// TwinCAT 3 PLC project Resolver_Test_Rig_Program
// ProgramVersion: 3.1.4023.0
// libraries:
//   Tc2_MC2, * (Beckhoff Automation GmbH)
//   Tc2_Standard, * (Beckhoff Automation GmbH)
//   Tc2_System, * (Beckhoff Automation GmbH)
//   Tc2_Utilities, * (Beckhoff Automation GmbH)
//   Tc3_Module, * (Beckhoff Automation GmbH)
//   VisuDialogs, * (System)
// project tree:
//   DUTs/ DUT_fileWriterStates.TcDUT, ST_EncoderCSVData.TcDUT
//   / GlobalTextList.TcGTLO, PlcTask.TcTTO, Visualization Manager.TcVMO (not stored)
//   GVLs/ GVL.TcGVL
//   POUs/ MAIN.TcPOU, FB_Stage_Motion.TcPOU, P_CSVWriter.TcPOU
//   POUs/UnixTimestamp/ UnixTimestamp.TcPOU (not stored)
//   VISUs/ Alarms.TcVIS, Manual_Operations.TcVIS, Run_Screen.TcVIS, Set_Up.TcVIS, Visualization.TcVIS
// real-time tasks:
//   TASK PlcTask: cycle T#10ms, priority 5, ADS port 350
// motion (NC):
//   TASK NC-Task 1 SAF: cycle T#2ms, priority 4, ADS port 501
//   TASK NC-Task 1 SVB: cycle T#10ms, priority 8, ADS port 511
//   AXIS Axis 1 (id 1)
//     Dynamic: AccelerationMaximum=375, DecelerationMaximum=375
//     Velo: SlowManual=0.5, FastManual=1, Maximum=50
//     OtherSettings: AllowMotionCmdToSlave=true
//     encoder EncType=4
//       EncPara: ScaleFactorNumerator=0.00015625, MaxCount=#x0000ffff
//         Inc: RefMode=2, RefSoftSyncMask=#x0000ffff
//     drive DrvType=24
//       Analog: VeloReferenz=20, TorqueScale=10, ScaleFactorActTorque=0.1
//       TimeComp: TaskDelayCycles=1
//     controller CtrType=1
//       CtrPara: PriorControlFactor=1
//         Observer: BandWidth=20
//   AXIS Axis 2 (id 2)
//     OtherSettings: AllowMotionCmdToSlave=true
//     encoder EncType=5
//       EncPara: ScaleFactorNumerator=0.5, ScaleFactorDenominator=65536, MaxCount=#xffffffff, ReferenceSystem=1
//     drive DrvType=5
//       Analog: TorqueScale=10, ScaleFactorActTorque=0.1
//       TimeComp: TaskDelayCycles=1
//     controller CtrType=1
//       CtrPara: PriorControlFactor=1
//         Observer: BandWidth=20
//   AXIS Axis 3 (id 3)
//     OtherSettings: AllowMotionCmdToSlave=true
//     encoder EncType=5
//       EncPara: ScaleFactorNumerator=2, ScaleFactorDenominator=4096, ReferenceSystem=1
//     drive DrvType=5
//       Analog: TorqueScale=10, ScaleFactorActTorque=0.1
//       TimeComp: TaskDelayCycles=1
//     controller CtrType=1
//       CtrPara: PriorControlFactor=1
//         Observer: BandWidth=20
//   AXIS Axis 4 (id 4)
//     OtherSettings: AllowMotionCmdToSlave=true
//     encoder EncType=29
//       EncPara: MaxCount=#xffffffff
//     drive DrvType=5
//       Analog: TorqueScale=10, ScaleFactorActTorque=0.1
//       TimeComp: TaskDelayCycles=1
//     controller CtrType=1
//       CtrPara: PriorControlFactor=1
//         Observer: BandWidth=20
// I/O:
//   DEVICE Device 1 (EtherCAT) (disabled), AmsNetId 130.246.57.106.2.1
//     Term 8 (EK1200) [EK1200-5000 EtherCAT Power supply (2A E-Bus)]
//       Term 9 (EL1008) [EL1008 8Ch. Dig. Input 24V, 3ms]
//       Term 10 (EL2808) [EL2808 8Ch. Dig. Output 24V, 0.5A]
//       Term 11 (EL7047) [EL7047 1Ch. Stepper motor output stage (50V, 5A)]
//       Term 12 (EL5002) [EL5002 2Ch. SSI Encoder]
//       Term 1 (EL5042) [EL5042 2Ch. BiSS-C Encoder]
//       Term 2 (EL3314-0002) [EL3314-0002 4Ch. Ana Input Thermocouple (TC), Isolated Channels]
//       Term 13 (EL9011) [EL9011 End Terminal]
// variable links:
//   NC-Task 1 SAF/Axes/Axis 1 <-> Device 1 (EtherCAT)/Term 8 (EK1200)/Term 11 (EL7047)
//     Drive/Inputs/In/nState1 @bit 3 <-> STM Status/Status/Error
//     Drive/Inputs/In/nState1 @bit 7 <-> STM Status/Status/Motor stall
//     Drive/Inputs/In/nState1 @bit 5 <-> STM Status/Status/Moving negative
//     Drive/Inputs/In/nState1 @bit 4 <-> STM Status/Status/Moving positive
//     Drive/Inputs/In/nState1 @bit 1 <-> STM Status/Status/Ready
//     Drive/Inputs/In/nState1 <-> STM Status/Status/Ready to enable
//     Drive/Inputs/In/nState1 @bit 6 <-> STM Status/Status/Torque reduced
//     Drive/Inputs/In/nState1 @bit 2 <-> STM Status/Status/Warning
//     Drive/Inputs/In/nState2 @bit 3 <-> STM Status/Status/Digital input 1
//     Drive/Inputs/In/nState2 @bit 4 <-> STM Status/Status/Digital input 2
//     Drive/Inputs/In/nState2 @bit 5 <-> STM Status/Status/Sync error
//     Drive/Inputs/In/nState2 @bit 7 <-> STM Status/Status/TxPDO Toggle
//     Drive/Inputs/In/nState4 @bit 1 <-> WcState/InputToggle
//     Drive/Inputs/In/nState4 <-> WcState/WcState
//     Drive/Outputs/Out/nCtrl1 <-> STM Control/Control/Enable
//     Drive/Outputs/Out/nCtrl1 @bit 2 <-> STM Control/Control/Reduce torque
//     Drive/Outputs/Out/nCtrl1 @bit 1 <-> STM Control/Control/Reset
//     Drive/Outputs/Out/nCtrl2 @bit 3 <-> STM Control/Control/Digital output 1
//     Drive/Outputs/Out/nDataOut2[0] <-> STM Velocity/Velocity
//     Enc/Inputs/In/nDataIn1[0] <-> ENC Status compact/Counter value
//     Enc/Inputs/In/nDataIn2[0] <-> ENC Status compact/Latch value
//     Enc/Inputs/In/nState1 @bit 4 <-> ENC Status compact/Status/Counter overflow
//     Enc/Inputs/In/nState1 @bit 3 <-> ENC Status compact/Status/Counter underflow
//     Enc/Inputs/In/nState1 @bit 7 <-> ENC Status compact/Status/Extrapolation stall
//     Enc/Inputs/In/nState1 <-> ENC Status compact/Status/Latch C valid
//     Enc/Inputs/In/nState1 @bit 1 <-> ENC Status compact/Status/Latch extern valid
//     Enc/Inputs/In/nState1 @bit 2 <-> ENC Status compact/Status/Set counter done
//     Enc/Inputs/In/nState2 @bit 4 <-> ENC Status compact/Status/Status of extern latch
//     Enc/Inputs/In/nState2 <-> ENC Status compact/Status/Status of input A
//     Enc/Inputs/In/nState2 @bit 1 <-> ENC Status compact/Status/Status of input B
//     Enc/Inputs/In/nState2 @bit 2 <-> ENC Status compact/Status/Status of input C
//     Enc/Inputs/In/nState2 @bit 5 <-> ENC Status compact/Status/Sync error
//     Enc/Inputs/In/nState2 @bit 7 <-> ENC Status compact/Status/TxPDO Toggle
//     Enc/Inputs/In/nState4 @bit 1 <-> WcState/InputToggle
//     Enc/Inputs/In/nState4 <-> WcState/WcState
//     Enc/Outputs/Out/nCtrl1 <-> ENC Control compact/Control/Enable latch C
//     Enc/Outputs/Out/nCtrl1 @bit 3 <-> ENC Control compact/Control/Enable latch extern on negative edge
//     Enc/Outputs/Out/nCtrl1 @bit 1 <-> ENC Control compact/Control/Enable latch extern on positive edge
//     Enc/Outputs/Out/nCtrl1 @bit 2 <-> ENC Control compact/Control/Set counter
//     Enc/Outputs/Out/nDataOut1[0] <-> ENC Control compact/Set counter value
//   NC-Task 1 SAF/Axes/Axis 2 <-> Device 1 (EtherCAT)/Term 8 (EK1200)/Term 12 (EL5002)
//     Enc/Inputs/In/nDataIn1 <-> SSI Inputs Channel 1/Counter value
//     Enc/Inputs/In/nState1 <-> SSI Inputs Channel 1/Status/Data error
//     Enc/Inputs/In/nState1 @bit 3 <-> SSI Inputs Channel 1/Status/Data mismatch
//     Enc/Inputs/In/nState1 @bit 1 <-> SSI Inputs Channel 1/Status/Frame error
//     Enc/Inputs/In/nState1 @bit 2 <-> SSI Inputs Channel 1/Status/Power failure
//     Enc/Inputs/In/nState2 @bit 5 <-> SSI Inputs Channel 1/Status/Sync error
//     Enc/Inputs/In/nState2 @bit 6 <-> SSI Inputs Channel 1/Status/TxPDO State
//     Enc/Inputs/In/nState2 @bit 7 <-> SSI Inputs Channel 1/Status/TxPDO Toggle
//     Enc/Inputs/In/nState4 @bit 1 <-> WcState/InputToggle
//     Enc/Inputs/In/nState4 <-> WcState/WcState
//   NC-Task 1 SAF/Axes/Axis 3 <-> Device 1 (EtherCAT)/Term 8 (EK1200)/Term 12 (EL5002)
//     Enc/Inputs/In/nDataIn1 <-> SSI Inputs Channel 2/Counter value
//     Enc/Inputs/In/nState1 <-> SSI Inputs Channel 2/Status/Data error
//     Enc/Inputs/In/nState1 @bit 3 <-> SSI Inputs Channel 2/Status/Data mismatch
//     Enc/Inputs/In/nState1 @bit 1 <-> SSI Inputs Channel 2/Status/Frame error
//     Enc/Inputs/In/nState1 @bit 2 <-> SSI Inputs Channel 2/Status/Power failure
//     Enc/Inputs/In/nState2 @bit 5 <-> SSI Inputs Channel 2/Status/Sync error
//     Enc/Inputs/In/nState2 @bit 6 <-> SSI Inputs Channel 2/Status/TxPDO State
//     Enc/Inputs/In/nState2 @bit 7 <-> SSI Inputs Channel 2/Status/TxPDO Toggle
//     Enc/Inputs/In/nState4 @bit 1 <-> WcState/InputToggle
//     Enc/Inputs/In/nState4 <-> WcState/WcState
//   NC-Task 1 SAF/Axes/Axis 4 <-> Device 1 (EtherCAT)/Term 8 (EK1200)/Term 1 (EL5042)
//     Enc/Inputs/In/nComState @bit 1 <-> WcState/InputToggle
//     Enc/Inputs/In/nComState <-> WcState/WcState
//     Enc/Inputs/In/nDataIn1 <-> FB Inputs Channel 1/Position
//     Enc/Inputs/In/nState1 @bit 12 <-> FB Inputs Channel 1/Status/Diag
//     Enc/Inputs/In/nState1 @bit 1 <-> FB Inputs Channel 1/Status/Error
//     Enc/Inputs/In/nState1 @bit 14 <-> FB Inputs Channel 1/Status/Input cycle counter
//     Enc/Inputs/In/nState1 @bit 2 <-> FB Inputs Channel 1/Status/Ready
//     Enc/Inputs/In/nState1 @bit 13 <-> FB Inputs Channel 1/Status/TxPDO State
//     Enc/Inputs/In/nState1 <-> FB Inputs Channel 1/Status/Warning
//   Resolver_Test_Rig_Program/Resolver_Test_Rig_Program Instance <-> Device 1 (EtherCAT)/Term 8 (EK1200)/Term 10 (EL2808)
//     PlcTask Outputs/MAIN.EncoderPowerOutput_3 <-> Channel 3/Output
//     PlcTask Outputs/MAIN.EncoderPowerOutput_6 <-> Channel 6/Output
//     PlcTask Outputs/MAIN.LimitSwitchOutput_1 <-> Channel 1/Output
//     PlcTask Outputs/MAIN.LimitSwitchOutput_2 <-> Channel 2/Output
//   Resolver_Test_Rig_Program/Resolver_Test_Rig_Program Instance <-> Device 1 (EtherCAT)/Term 8 (EK1200)/Term 9 (EL1008)
//     PlcTask Inputs/MAIN.LimitSwitchInput_1 <-> Channel 1/Input
//     PlcTask Inputs/MAIN.LimitSwitchInput_2 <-> Channel 2/Input

CONFIGURATION Resolver_Test_Rig_Program
    RESOURCE PLC ON TwinCAT3
        TASK PlcTask(INTERVAL := T#10ms, PRIORITY := 5);
        PROGRAM MAIN WITH PlcTask : MAIN;
    END_RESOURCE
END_CONFIGURATION

// ---- DUTs/DUT_fileWriterStates.TcDUT
{attribute 'qualified_only'}
{attribute 'strict'}
TYPE DUT_fileWriterStates :
(
	
    idle := 0,
    opening,
    saving,
    closing,
    error

);
END_TYPE

// ---- DUTs/ST_EncoderCSVData.TcDUT
TYPE ST_EncoderCSVData :
STRUCT
	MeasurementID           : INT;
    testState               : INT;
    AxisPosition            : LREAL;
    CurrentCycle            : WORD;
    PositalPosition         : LREAL;
    KublerPosition          : LREAL;
    AMOPosition             : REAL;
    ThermoCouple            : ARRAY[0..3] OF DINT;
    UnixTime                : ULINT;
END_STRUCT
END_TYPE

// ---- GVLs/GVL.TcGVL
{attribute 'Tc2GvlVarNames'}
VAR_GLOBAL CONSTANT
	

	MAX_CSV_ROWS             : UDINT := 1;
    MAX_CSV_COLUMNS         : UDINT := 12;
    MAX_CSV_FIELD_LENGTH    : UDINT := 100;
   
    DATA_CSV_HEADERS        : ARRAY[0..MAX_CSV_COLUMNS] OF STRING(MAX_CSV_FIELD_LENGTH) :=[ (* Source PLC database *)
    'MeasurementID',
    'TestState',
    'AxisPosition',
    'CurrentCycle',
    'PositalPosition',
    'KublerPosition',
    'AMOPosition',
    'ThermoCouple_1',
    'ThermoCouple_2',
    'ThermoCouple_3',
    'ThermoCouple_4',  
    'UnixTime']; 

END_VAR 
VAR_GLOBAL
		stAxis_1 : AXIS_REF;
		stAxis_2 : AXIS_REF;
		stAxis_3 : AXIS_REF;
		stAxis_4 : AXIS_REF;
		

END_VAR

// ---- POUs/MAIN.TcPOU
PROGRAM MAIN
VAR
		// stepper function blocks  
	mcPower_1 : MC_Power;
	mcReset_1 : MC_Reset;
	mcJogging_1 : MC_Jog;
	mcMoveAbs_1 : MC_MoveAbsolute;
	mcMoveRel_1 : MC_MoveRelative;
	mcStop : MC_Stop;
	mcHome_1 : MC_Home;
	
	bEnableAxis_1 : BOOL;
	bJogForwards : BOOL;
	bJogBackwards: BOOL;
	eJogMode : E_JogMode; 
	bMoveDone : BOOL;	
	bAbsMove: BOOL;
	bRelMove: BOOL;
	
	heartbeat: BYTE; 
	//FbStageMotion : FB_Stage_Motion;

	bStop: BOOL;
	bHomeAxis_1: BOOL;

	// action Variables
	mcMoveAbsTest_1 : MC_MoveAbsolute;
	mcMoveAbsTestReturn_1 : MC_MoveAbsolute;
	iState : DINT;
	bStartTest : BOOL;
	bFinishTest: BOOL;
	fbReturnTimer : TON; // timer delay for the cycle to return home.
	fbDutyCycleTimer : TON; // timer duty cycle so the delay between cycles
	bStartReturnTimer : BOOL;
	bStartDutyCycleTimer : BOOL;	
	fbTestCycleCounter  : CTU;
	bCycleComplete : BOOL;
	bCycleCounterReset : BOOL;
	bTestFinished : BOOL;
	bTestRelMove: BOOL;
	

	bEnableAxisPosative_1: BOOL;
	bEnableAxisNegative_1: BOOL;
END_VAR

VAR_INPUT
	fAbsPos_1: LREAL;
	fRelDistance: LREAL;
	fRelTestDistance: LREAL;
	fAbsTestDistance: LREAL;
	fHomePosition: LREAL;
	fAxisVelocity: LREAL;
	fAxisAcceleration: LREAL;
	// action Variables
	iCycleCount : WORD;
	fReturnTime: TIME;
	uInputReurnTime :UDINT;
	fDutyCycleTime: TIME;
	uInputCycleTime :UDINT;
	
			// Digital Inputs
	LimitSwitchInput_1 AT %I* : BOOL;
	LimitSwitchInput_2 AT %I* : BOOL;
			// Analogue inputs
	ThermoCoupleChannel_1 AT %I*: REAL;
	ThermoCoupleChannel_2 AT %I*: REAL;
	ThermoCoupleChannel_3 AT %I*: REAL;
	ThermoCoupleChannel_4 AT %I*: REAL;
END_VAR

VAR_OUTPUT
// action Variables	
	iCurrentCycleValue : WORD;
		// Digital outputs
	LimitSwitchOutput_1 AT %Q* : BOOL;
	LimitSwitchOutput_2 AT %Q* : BOOL;
	EncoderPowerOutput_3 AT %Q* : BOOL;
	EncoderPowerOutput_6 AT %Q* : BOOL;
END_VAR

heartbeat := heartbeat + 1;

Limit_Switch();
EncoderPowerOutput_3 := TRUE;
EncoderPowerOutput_6 := TRUE;

mcStop(Axis := GVL.stAxis_1, Execute := bStop,);

mcPower_1(Axis := GVL.stAxis_1, Enable := bEnableAxis_1, Enable_Positive := bEnableAxisPosative_1, Enable_Negative := bEnableAxisNegative_1, Override := 100.0);

mcReset_1(Axis := GVL.stAxis_1, Execute := NOT(bEnableAxis_1));

mcJogging_1(Axis := GVL.stAxis_1, JogForward := bJogForwards, JogBackwards := bJogBackwards, Velocity := fAxisVelocity, Acceleration := fAxisAcceleration, Deceleration := fAxisAcceleration, Jerk := 0.8);

mcMoveAbs_1 (Axis := GVL.stAxis_1, Execute := bAbsMove, Position := fAbsPos_1, Velocity := fAxisVelocity, Acceleration := fAxisAcceleration, Deceleration := fAxisAcceleration);
bAbsMove := FALSE;

mcMoveRel_1(Axis := GVL.stAxis_1, Execute := bRelMove, Distance := fRelDistance, Velocity := fAxisVelocity, Acceleration := fAxisAcceleration, Deceleration := fAxisAcceleration);
bRelMove := FALSE;

//mcHome_1(Axis := GVL.stAxis_1, Execute := bHomeAxis_1, Position := fHomePosition);

Test_Routine();

P_CSVWriter(     bNewData            :=    TRUE);

ACTION Limit_Switch:
LimitSwitchOutput_1 := TRUE;
LimitSwitchOutput_2 := TRUE;

IF LimitSwitchInput_1 THEN
	bEnableAxisPosative_1 := TRUE;
ELSE
	bEnableAxisPosative_1 := FALSE ;	
	
END_IF

IF LimitSwitchInput_2 THEN
	bEnableAxisNegative_1 := TRUE;
ELSE
	bEnableAxisNegative_1 := FALSE ;	
	
END_IF
END_ACTION

ACTION Test_Routine:
mcMoveAbsTest_1(Axis := GVL.stAxis_1, Position := 10, Velocity := fAxisVelocity, Acceleration := fAxisAcceleration, Deceleration := fAxisAcceleration);	
mcMoveAbsTest_1.Execute := FALSE;
fbReturnTimer( IN := bStartReturnTimer, PT := fReturnTime);	
mcMoveAbsTestReturn_1(Axis := GVL.stAxis_1, Position := 0, Velocity := fAxisVelocity, Acceleration := fAxisAcceleration, Deceleration := fAxisAcceleration);
mcMoveAbsTestReturn_1.Execute := FALSE;
fbReturnTimer( IN := bStartReturnTimer, PT := fReturnTime);	
fbDutyCycleTimer( IN := bStartDutyCycleTimer, PT := fDutyCycleTime);	
fbTestCycleCounter(CU := bCycleComplete, RESET := bCycleCounterReset, PV := iCycleCount);
fReturnTime:= UDINT_TO_TIME(uInputReurnTime);
fDutyCycleTime:= UDINT_TO_TIME(uInputCycleTime);
CASE iState OF
	
	// initialising the state machine so starting a homing rotuine reseting the counter to 0 
	0: 
		iState := 10;
	10: 
		IF bStartTest THEN
			P_CSVWriter(bOpen:=TRUE);
			iState := 20;
		END_IF
	
	20:
		
		mcMoveAbsTest_1.Execute := TRUE;
		IF mcMoveAbsTest_1.Done THEN
			bStartReturnTimer := TRUE;
			iState := 30;
		END_IF

	30:
		fbReturnTimer( IN := bStartReturnTimer, PT := fReturnTime);	
		IF MAIN.fbReturnTimer.Q THEN
			bStartReturnTimer := FALSE;
			iState := 40;
		END_IF
	

	40:
		mcMoveAbsTestReturn_1.Execute := TRUE;
		IF mcMoveAbsTestReturn_1.Done THEN
			bStartDutyCycleTimer := TRUE;
			iState := 50;
		END_IF	
	
	50:
		fbDutyCycleTimer( IN := bStartDutyCycleTimer, PT := fDutyCycleTime);	
		IF MAIN.fbDutyCycleTimer.Q THEN
			bStartDutyCycleTimer := FALSE;
			iState := 60;
		END_IF

	60: bCycleComplete := TRUE;
		iState := 70;
	
	70: fbTestCycleCounter(CU := bCycleComplete, RESET := bCycleCounterReset, PV := iCycleCount);
		IF MAIN.fbTestCycleCounter.Q THEN
			iState := 90; 
		ELSE
		bCycleComplete := FALSE;	
		iState := 20;
		END_IF
	
	90: bStartTest := FALSE;
		bFinishTest := TRUE;
		P_CSVWriter(bClose   :=  TRUE);
		iState := 10;
	
ELSE
	;
END_CASE
END_ACTION

ACTION Thermo_Couple:
IF ThermoCoupleChannel_1 > 40 THEN
	bEnableAxis_1 := FALSE ;
		
	
END_IF

IF ThermoCoupleChannel_2 > 40 THEN
	bEnableAxis_1 := FALSE ;
		
	
END_IF
END_ACTION

END_PROGRAM

// ---- POUs/P_CSVWriter.TcPOU
PROGRAM P_CSVWriter
(* Writing of CSV file in text mode. None of the field value is containing any non-printing control characters like line feed, carriage return, quotation marks, semicolon... *)
VAR
	
	bBusy			: BOOL := TRUE;
	
	
	sNetId			: T_AmsNetId := '';	(* TwinCAT system network address *)
	sFileName		: T_MaxString := 'C:\ShutterTestData\';(* CSV destination file path and name *)
	sCSVLine		: T_MaxString := '';(* Single CSV text line (row, record), we are using string as record buffer (your are able to see created fields) *)
	
	
	nErrId			: UDINT;
	
	//File management fucntion blocks and variables
	fbWriter		: FB_CSVMemBufferWriter;(* Helper function block used to create CSV data bytes (single record line) *)
	hFile			: UINT		:= 0;(* File handle of the source file *)
	step			: DWORD 	:= 0;
	fbFileOpen		: FB_FileOpen;(* Opens file *)
	fbFileClose		: FB_FileClose;(* Closes file *)
	fbFilePuts		: FB_FilePuts;(* Writes one record (line) *)
	
	//UnixTimestamp function block
	unixTime: UnixTimestamp;
    timestampMilliseconds: ULINT;
	
	//State Mechine
	dataWriterState 		: DUT_fileWriterStates := DUT_fileWriterStates.idle;
	
	//Timer for when to save
	saveIntervalTimer		: TON;
	
END_VAR
VAR_INPUT
	//test data//
	testEncoderData : ST_EncoderCSVData;
	
	bNewData		: BOOL := FALSE;	(* Rising edge starts data saving*)
	bOpen			: BOOL := FALSE;	(* Rising edge starts program execution *)
	bClose			: BOOL := FALSE;	(* Rising edge ends program execution *)
	
	
	saveInterval	: TIME := T#100MS;
	
	stimeString		: T_MaxString;
END_VAR
VAR_OUTPUT
	//Error flag for troubleshooting
	bError			: BOOL;
	
	//Mesurement ID 
	nMeasurementID	: INT := 0;
END_VAR

CASE dataWriterState OF
	DUT_fileWriterStates.idle:	(* Wait for rising edge at bOpen variable *)
		nMeasurementID := 0;
		
		
		//Check of rising edge on open boolean
		IF bOpen THEN
			dataWriterState := DUT_fileWriterStates.opening;
		END_IF
		
		//"Opening State" initalisation code
		//reset variables (incase the PLC has not been reset
		IF dataWriterState = DUT_fileWriterStates.opening THEN
			bOpen 					:= FALSE;
			bClose					:= FALSE;
			
			bBusy					:= TRUE;
			bError					:= FALSE;
			nErrId					:= 0;
			hFile					:= 0;
			
			//Set the seperator to be a comma
			DEFAULT_CSV_FIELD_SEP := 16#2C;
			
			//start opening file
			OpenFile();
		END_IF
	
	//Stay this state until file has been opened
	DUT_fileWriterStates.opening:	(* Wait until open not busy *)
		nMeasurementID := 0;
		//Check if the file opening has been complete
		IF CheckIfOpened() THEN			
			dataWriterState := DUT_fileWriterStates.saving;(* Write record to the file *)
		END_IF
		
		
		
		//If state has been changed to saving, the headers for the data are applied to the top of the CSV
		IF dataWriterState = DUT_fileWriterStates.saving THEN
			WriteCSVLine(StringArrayToCSVString(DATA_CSV_HEADERS));	
		END_IF
	
	//Save data until rising edge on bclose variables
	DUT_fileWriterStates.saving: 
		(* Wait for rising edge at bNewData variable *)
		saveIntervalTimer(IN := TRUE, PT := saveInterval);
		IF bNewData AND saveIntervalTimer.Q THEN
			//reset save interval timer
			saveIntervalTimer(IN := FALSE);
			//save and increment measurement ID
			testEncoderData.MeasurementID := nMeasurementID;
			nMeasurementID := nMeasurementID + 1;
			//Write shuitter data to CSV
			WriteCSVLine(EncoderDataToCSVString(testEncoderData));
			bNewData := FALSE;
		END_IF
		
		(* Wait for rising edge at bClose variable *)
		IF bClose THEN
			dataWriterState := DUT_fileWriterStates.closing;
		END_IF
		//Close the file before moving onto the closing state
		IF dataWriterState = DUT_fileWriterStates.closing THEN
			bClose := FALSE; 
			CloseFile();
			
			//reset measurement ID
			nMeasurementID:= 0;
		END_IF
		
	DUT_fileWriterStates.closing:	(* Close source file *)
		IF CheckIfClosed() THEN
			dataWriterState := DUT_fileWriterStates.idle;	(* Ready *)
		END_IF
		
		
	DUT_fileWriterStates.error: (* Error detected TODO:  *)
		bError := TRUE;
END_CASE

//Check if an error has occured
IF bError THEN
	dataWriterState := DUT_fileWriterStates.error;
END_IF

METHOD CheckIfClosed : BOOL
VAR_INPUT
END_VAR
fbFileClose( bExecute := FALSE, bError => bError, nErrID => nErrID );
IF ( NOT fbFileClose.bBusy ) THEN
			hFile := 0;
			CheckIfClosed := TRUE;
ELSE
				
			CheckIfClosed := FALSE;
			
END_IF
END_METHOD

METHOD CheckIfOpened : BOOL
VAR_INPUT
END_VAR
VAR_OUTPUT
	errorOpening : BOOL := FALSE;
END_VAR
fbFileOpen( bExecute := FALSE, bError => bError, nErrID => nErrID, hFile => hFile );
IF NOT fbFileOpen.bBusy THEN
	IF NOT fbFileOpen.bError THEN
		CheckIfOpened := TRUE;
	ELSE(* Error: file not found? *)
		errorOpening := TRUE;
	END_IF
ELSE
	CheckIfOpened := FALSE;
END_IF
END_METHOD

METHOD CloseFile : BOOL
VAR_INPUT
END_VAR
fbFileClose( bExecute := FALSE );
fbFileClose( sNetId := sNetId, hFile := hFile, bExecute := TRUE );
END_METHOD

METHOD EncoderDataToCSVString : T_MaxString
VAR_INPUT
	inputEncoderData : ST_EncoderCSVData;
END_VAR

VAR_OUTPUT
	tempArray	: ARRAY[0..MAX_CSV_COLUMNS] OF STRING(MAX_CSV_FIELD_LENGTH);
END_VAR

VAR
	
END_VAR

tempArray := EncoderDataToStringArray(inputEncoderData);
EncoderDataToCSVString := StringArrayToCSVString(tempArray);
END_METHOD

METHOD EncoderDataToStringArray :  ARRAY[0..MAX_CSV_COLUMNS] OF STRING(MAX_CSV_FIELD_LENGTH);
VAR_INPUT
	inputEncoderData : ST_EncoderCSVData;
END_VAR
EncoderDataToStringArray[0] := INT_TO_STRING(inputEncoderData.MeasurementID);
EncoderDataToStringArray[1] := INT_TO_STRING(inputEncoderData.testState);
EncoderDataToStringArray[2] := LREAL_TO_STRING(inputEncoderData.AxisPosition);
EncoderDataToStringArray[3] := WORD_TO_STRING(inputEncoderData.CurrentCycle);
EncoderDataToStringArray[4] := LREAL_TO_STRING(inputEncoderData.PositalPosition);
EncoderDataToStringArray[5] := LREAL_TO_STRING(inputEncoderData.KublerPosition);
EncoderDataToStringArray[6] := LREAL_TO_STRING(inputEncoderData.AMOPosition);
EncoderDataToStringArray[7] := DINT_TO_STRING(inputEncoderData.ThermoCouple[0]);
EncoderDataToStringArray[8] := DINT_TO_STRING(inputEncoderData.ThermoCouple[1]);
EncoderDataToStringArray[9] := DINT_TO_STRING(inputEncoderData.ThermoCouple[2]);
EncoderDataToStringArray[10] := DINT_TO_STRING(inputEncoderData.ThermoCouple[3]);
EncoderDataToStringArray[11] := ULINT_TO_STRING(inputEncoderData.UnixTime);
END_METHOD

METHOD OpenFile : BOOL
VAR_INPUT
END_VAR
VAR
	fbCreateDir	: FB_CreateDir;	


	newPath : STRING(255);
	newPath2: STRING(255);
	sCSV	: STRING(255) := 'Test.csv';
END_VAR
//create directory
fbCreateDir(bExecute := FALSE);
fbCreateDir(
		sNetId := '',
		sPathName := sFileName,
		ePath  := PATH_GENERIC,
		bExecute := TRUE,
		tTimeout := DEFAULT_ADS_TIMEOUT);
		
//open file
fbFileOpen(  bExecute := FALSE  );

stimeString := REPLACE(stimeString,'.',1,5);
stimeString := REPLACE(stimeString,'.',1,8);
stimeString := REPLACE(stimeString,'.',1,11);
stimeString := REPLACE(stimeString,'.',1,14);
stimeString := REPLACE(stimeString,'.',1,17);
newPath := CONCAT(sFileName,stimeString);
newPath2:= CONCAT(newPath,sCSV);

fbFileOpen( 	sNetId := sNetId, 
				sPathName := newPath2, 
				nMode := FOPEN_MODEWRITE OR FOPEN_MODETEXT,(* Open file in TEXT mode! *)
				ePath := PATH_GENERIC,
				bExecute := TRUE );
END_METHOD

METHOD StringArrayToCSVString : T_MaxString
VAR_INPUT
	inputArray	: ARRAY[0..MAX_CSV_COLUMNS] OF STRING(MAX_CSV_FIELD_LENGTH);
END_VAR
VAR_OUTPUT
	
END_VAR
VAR
	nColumn		: UDINT 	:= 0;(* Column number (record field) *)
	sCSVField		: T_MaxString := '';(* Single CSV field value (column, record field) *)
	tempString		: T_MaxString := '';
	
	
END_VAR

FOR nColumn := 0 TO MAX_CSV_COLUMNS BY 1 DO

	sCSVField := STRING_TO_CSVFIELD( inputArray[ nColumn ], FALSE );(* TODO: Get field value from your application *)

				(* Add new field to the record buffer *)
	fbWriter( 	pBuffer := ADR( tempString ), cbBuffer := SIZEOF( tempString ) - 1, putValue := sCSVField, pValue := 0, cbValue := 0,
				bCRLF := ( nColumn = MAX_CSV_COLUMNS ) );(* bCRLF == TRUE => Write CRLF after the last field value *)
	IF fbWriter.bOk THEN
		fbWriter.eCmd := eEnumCmd_Next;(* Write next field value *)
	END_IF

END_FOR(* FOR nColumn := 0... *)

(* FB_FilePuts adds allready CR (carriage return) to the written line.
We have to replace the $R$L characters with $L character to avoid double CR. *)
IF RIGHT( tempString, 2 ) = '$R$L' THEN
	tempString := REPLACE( tempString, '$L', 2, LEN(tempString  ) - 1 );
END_IF

StringArrayToCSVString := tempString;
END_METHOD

METHOD WriteCSVLine : BOOL
VAR_INPUT
	newSCVLine : T_MAXSTRING;
END_VAR
VAR
	canSave		: BOOL :=FALSE;
END_VAR
fbFilePuts( bExecute := FALSE, bError => bError, nErrID => nErrID );
IF NOT fbFilePuts.bBusy THEN
	IF NOT fbFilePuts.bError THEN
		canSave := TRUE;
	ELSE(* Error *)
		//dataWriterState := DUT_fileWriterStates.error;
	END_IF
END_IF


IF canSave THEN
			fbWriter.eCmd := eEnumCmd_First;
			fbFilePuts( bExecute := FALSE );
			fbFilePuts( sNetId := sNetId, hFile := hFile, sLine := newSCVLine, bExecute := TRUE );
			//dataWriterState := DUT_fileWriterStates.saving;(* Write record to the file *)
END_IF
END_METHOD

END_PROGRAM

// ---- POUs/FB_Stage_Motion.TcPOU
FUNCTION_BLOCK FB_Stage_Motion
VAR_INPUT

END_VAR
VAR_OUTPUT
END_VAR
VAR
		// stepper function blocks  
	mcPower_1 : MC_Power;
	mcReset_1 : MC_Reset;
	mcJogging_1 : MC_Jog;
	mcMoveAbs_1 : MC_MoveAbsolute;
	mcMoveRel_1 : MC_MoveRelative;
	
	bEnableAxis_1 : BOOL;
	bJogForwards : BOOL;
	eJogMode : E_JogMode; 
	bMoveDone : BOOL;	
	bAbsMove: BOOL;
	fAbsPos_1: LREAL;
	bRelMove: BOOL;
	fRelDistance: LREAL;
END_VAR

mcPower_1(Axis := GVL.stAxis_1, Enable := bEnableAxis_1, Enable_Positive := TRUE, Enable_Negative := TRUE, Override := 100.0);

mcReset_1(Axis := GVL.stAxis_1, Execute := NOT(bEnableAxis_1));

mcJogging_1(Axis := GVL.stAxis_1, JogForward := bJogForwards, Mode := MC_JOGMODE_INCHING, Position := 360.0, Velocity := 1.0, Acceleration := 1.0, Deceleration := 1.0, Jerk := 0.8);

mcMoveAbs_1 (Axis := GVL.stAxis_1, Execute := bAbsMove, Position := fAbsPos_1, Velocity := 1);

mcMoveRel_1(Axis := GVL.stAxis_1, Execute := bRelMove, Distance := fRelDistance, Velocity :=1);

END_FUNCTION_BLOCK

// ---- GlobalTextList.TcGTLO
TEXTLIST GlobalTextList
  816 = ' %i Cycles'
  217 = '%.0f '
  441 = '%.0f mS'
  934 = '%.1f mm/s'
  199 = '%.1f mm/s^2'
  229 = '%.1f mS'
  330 = '%.1s mS'
  618 = '%.2f mm'
  31 = '%.3f mm'
  39 = '%0.0f'
  20 = '%0.F'
  327 = '%0.f'
  498 = '%0.f mS'
  409 = '%F'
  933 = '%f'
  789 = '%f mm'
  608 = '%f mS'
  206 = '%f..2 mm'
  481 = '%f.2 mm'
  735 = '%i Cycles'
  12 = '%I mm'
  32 = '%i mm'
  540 = '%i mS'
  766 = '%R mm'
  590 = '%s'
  489 = '%s mm'
  744 = '%S mm'
  918 = '%t mS'
  802 = '%w mS'
  968 = 'Alarms'
  989 = 'AMO Position'
  974 = 'Axis Acceleration'
  630 = 'Axis Enable'
  44 = 'Axis Position'
  690 = 'Axis Speed'
  501 = 'Curret Cycle'
  78 = 'Cycle No. %i'
  542 = 'Delay Between Cycles'
  681 = 'Delay Between moves'
  336 = 'Jog Backwards'
  673 = 'Jog Forwards'
  242 = 'Kubler Position'
  60 = 'Manual Operations'
  410 = 'Move Absolute'
  811 = 'Move Relative'
  5 = 'No. Of Test Cycles'
  891 = 'Posital Position'
  653 = 'Position'
  146 = 'RESET'
  149 = 'Run Screen'
  19 = 'Set Up'
  478 = 'Setup'
  825 = 'Setup Screen'
  577 = 'Start Test'
  603 = 'STOP'
  898 = 'Test cycle'
  900 = 'Test cycles'
END_TEXTLIST

// ---- VISUs/Alarms.TcVIS
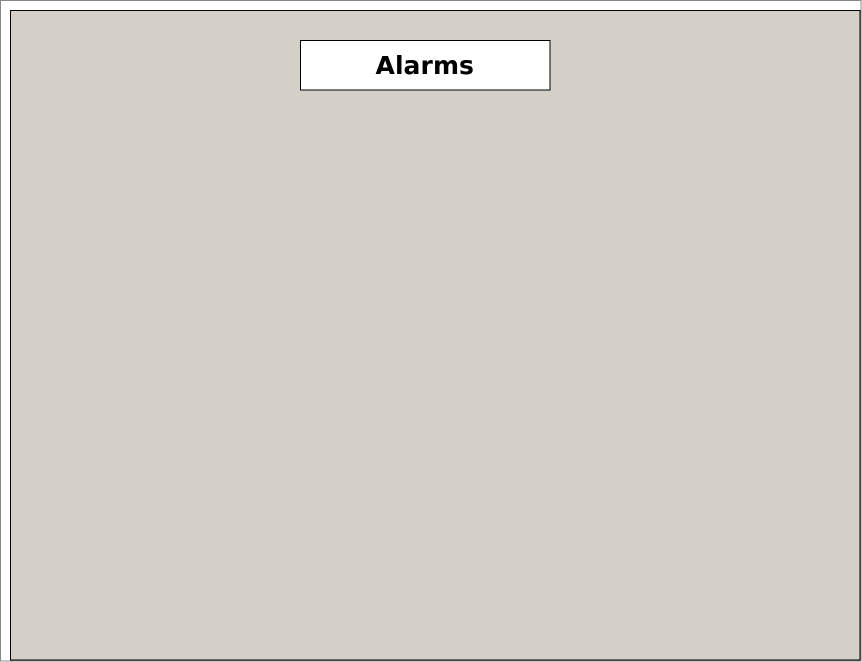
VISUALIZATION Alarms  // 862x662
    RoundedRectangle (10,10 850x650)
    RoundedRectangle (300,40 250x50), "Alarms"
END_VISUALIZATION

// ---- VISUs/Manual_Operations.TcVIS
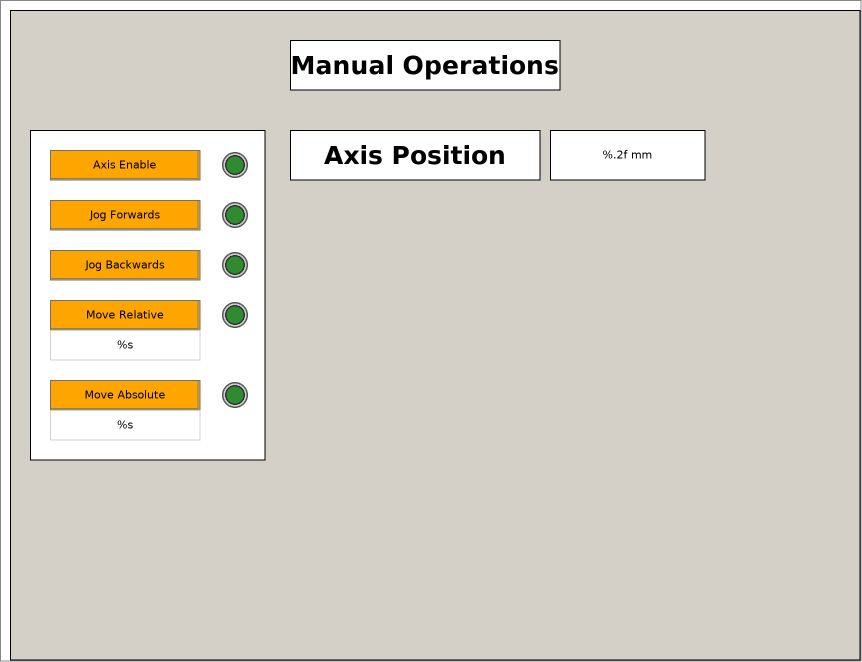
VISUALIZATION Manual_Operations  // 862x662
    RoundedRectangle (10,10 850x650)
    Rectangle (30,130 235x330)
    RoundedRectangle (290,40 270x50), "Manual Operations"
    Button (50,200 150x30), "Jog Forwards"
        OnMouseDown: toggle MAIN.bJogForwards
        OnMouseUp: toggle MAIN.bJogForwards
        OnMouseUp: execute { MAIN.bEnableAxis_1 := TRUE }
    Lamp1 (220,200 30x30), variable: MAIN.bJogForwards, style: Lamp-Lamp1-Green
    Button (50,150 150x30), "Axis Enable"
        toggle MAIN.bEnableAxis_1
    Lamp1 (220,150 30x30), variable: MAIN.mcPower_1.Enable, style: Lamp-Lamp1-Green
    Button (50,250 150x30), "Jog Backwards"
        OnMouseDown: toggle MAIN.bJogBackwards
        OnMouseUp: toggle MAIN.bJogBackwards
        OnMouseUp: execute { MAIN.bEnableAxis_1 := TRUE }
    Lamp1 (220,250 30x30), variable: MAIN.bJogBackwards, style: Lamp-Lamp1-Green
    Button (50,300 150x30), "Move Relative"
        toggle MAIN.bRelMove p2164770859=TRUE
    Lamp1 (220,300 30x30), variable: MAIN.mcMoveRel_1.Active, style: Lamp-Lamp1-Green
    Textfield (50,330 150x30), "%s", text variable: MAIN.fRelDistance
        OnMouseClick: write the text variable via VisuDialogs.Numpad, min -100, max 100, format Relative Move Distance
    Button (50,380 150x30), "Move Absolute"
        toggle MAIN.bAbsMove p2164770859=TRUE
    Lamp1 (220,380 30x30), variable: MAIN.mcMoveAbs_1.Active, style: Lamp-Lamp1-Green
    Textfield (50,410 150x30), "%s", text variable: MAIN.fAbsPos_1
        OnMouseClick: write the text variable via VisuDialogs.Numpad, min -100, max 100, format Relative Move Distance
    RoundedRectangle (290,130 250x50), "Axis Position"
    RoundedRectangle (550,130 155x50), "%.2f mm", text variable: GVL.stAxis_1.NcToPlc.SetPos
END_VISUALIZATION

// ---- VISUs/Run_Screen.TcVIS
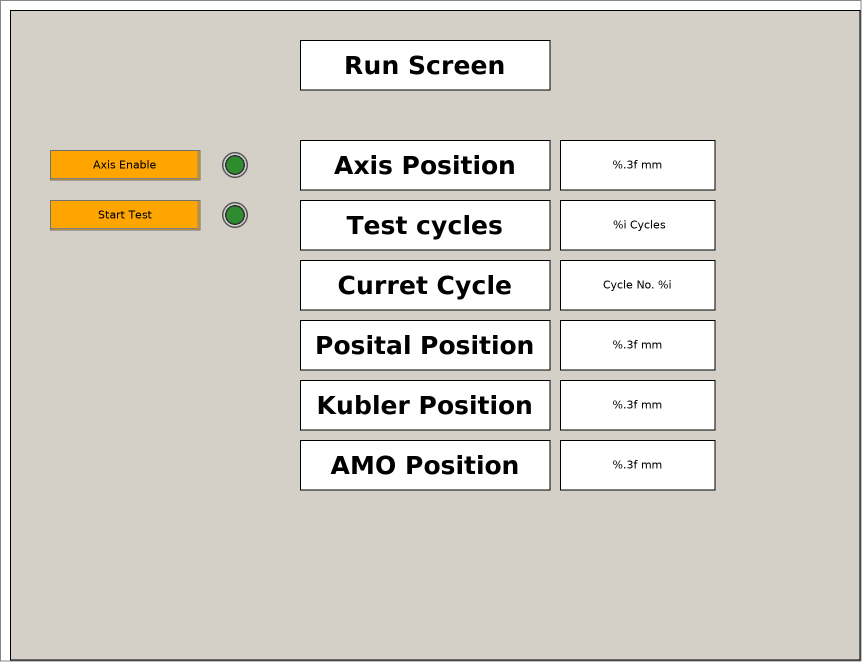
VISUALIZATION Run_Screen  // 862x662
    RoundedRectangle (10,10 850x650)
    RoundedRectangle (300,40 250x50), "Run Screen"
    Button (50,150 150x30), "Axis Enable"
        toggle MAIN.bEnableAxis_1
    Lamp1 (220,150 30x30), variable: MAIN.mcPower_1.Enable, style: Lamp-Lamp1-Green
    RoundedRectangle (300,140 250x50), "Axis Position"
    RoundedRectangle (560,140 155x50), "%.3f mm", text variable: GVL.stAxis_1.NcToPlc.SetPos
    RoundedRectangle (300,200 250x50), "Test cycles"
    RoundedRectangle (300,260 250x50), "Curret Cycle"
    RoundedRectangle (560,200 155x50), "%i Cycles", text variable: MAIN.fbTestCycleCounter.PV
    RoundedRectangle (560,260 155x50), "Cycle No. %i", text variable: MAIN.fbTestCycleCounter.CV
    Button (50,200 150x30), "Start Test"
        toggle MAIN.bStartTest
    Lamp1 (220,200 30x30), variable: MAIN.bStartTest, style: Lamp-Lamp1-Green
    RoundedRectangle (300,440 250x50), "AMO Position"
    RoundedRectangle (300,380 250x50), "Kubler Position"
    RoundedRectangle (300,320 250x50), "Posital Position"
    RoundedRectangle (560,380 155x50), "%.3f mm", text variable: stAxis_3.NcToPlc.ActPos
    RoundedRectangle (560,440 155x50), "%.3f mm", text variable: stAxis_4.NcToPlc.ActPos
    RoundedRectangle (560,320 155x50), "%.3f mm", text variable: stAxis_2.NcToPlc.ActPos
END_VISUALIZATION

// ---- VISUs/Set_Up.TcVIS
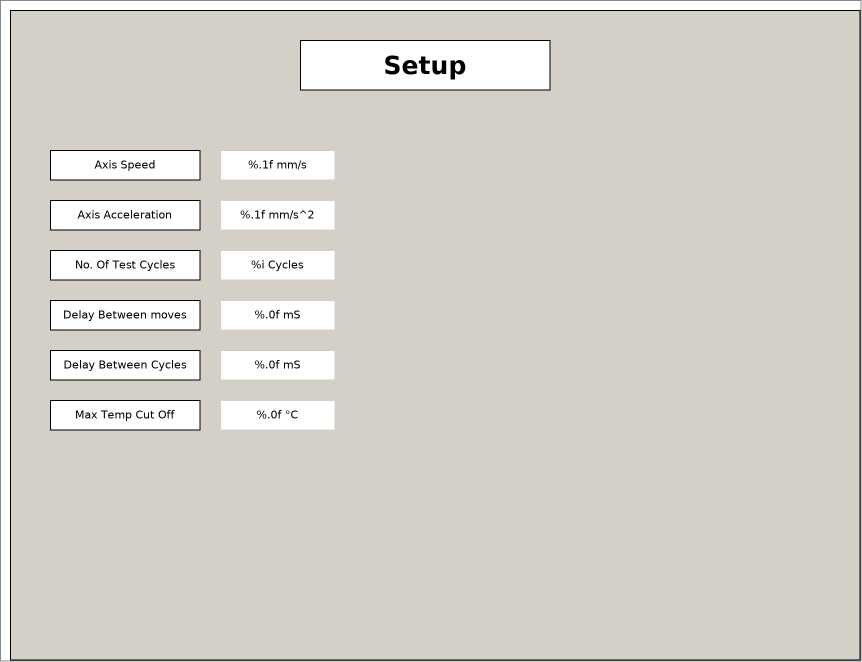
VISUALIZATION Set_Up  // 862x662
    RoundedRectangle (10,10 850x650)
    RoundedRectangle (300,40 250x50), "Setup"
    Rectangle (50,150 150x30), "Axis Speed"
    Textfield (220,150 115x30), "%.1f mm/s", text variable: MAIN.fAxisVelocity
        OnMouseClick: write the text variable via VisuDialogs.Numpad, min 0, max 20, format 1
    Rectangle (50,200 150x30), "Axis Acceleration"
    Textfield (220,200 115x30), "%.1f mm/s^2", text variable: MAIN.fAxisAcceleration
        OnMouseClick: write the text variable via VisuDialogs.Numpad, min 0, max 20, format 1
    Rectangle (50,350 150x30), "Delay Between Cycles"
    Rectangle (50,300 150x30), "Delay Between moves"
    Rectangle (50,250 150x30), "No. Of Test Cycles"
    Textfield (220,350 115x30), "%.0f mS", text variable: MAIN.uInputCycleTime
        OnMouseClick: write the text variable via VisuDialogs.Numpad
    Textfield (220,300 115x30), "%.0f mS", text variable: MAIN.uInputReurnTime
        OnMouseClick: write the text variable via VisuDialogs.Numpad
    Textfield (220,250 115x30), "%i Cycles", text variable: MAIN.iCycleCount
        OnMouseClick: write the text variable via VisuDialogs.Numpad, min 1, max 32000
    Rectangle (50,400 150x30), "Max Temp Cut Off"
    Textfield (220,400 115x30), "%.0f °C", text variable: MAIN.fTempLimit
        OnMouseClick: write the text variable via VisuDialogs.Numpad
END_VISUALIZATION

// ---- VISUs/Visualization.TcVIS
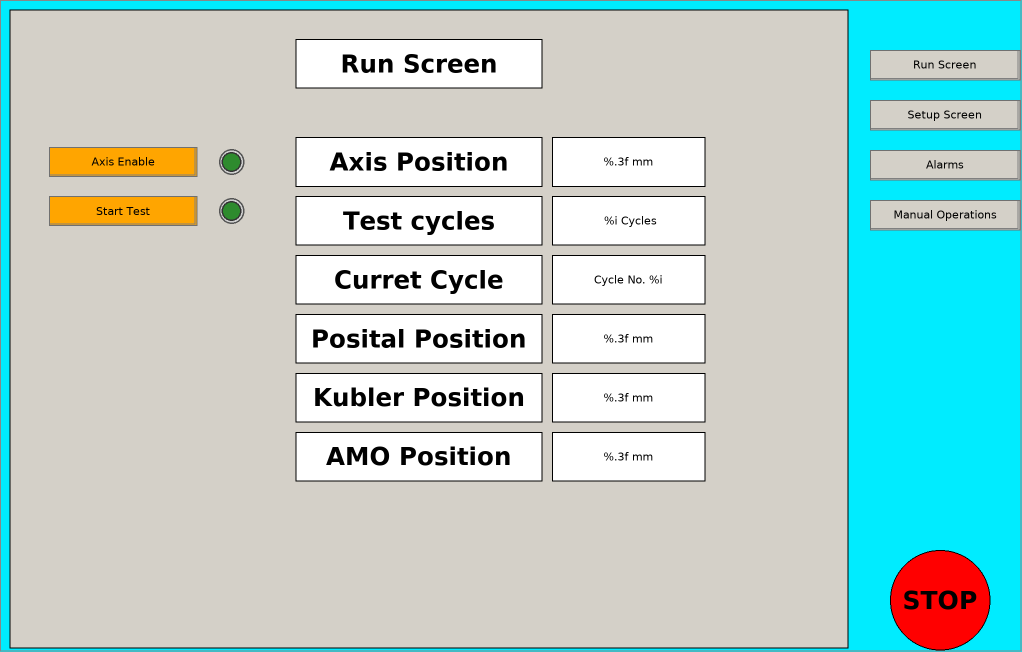
VISUALIZATION Visualization  // 1022x652
    Frame (0,0 850x650)
        shows Run_Screen()
        shows Set_Up()
        shows Alarms()
        shows Manual_Operations()
    Button (870,50 150x30), "Run Screen"
        OnMouseClick: FrameSelectionChange Selection=SelectedFrame=ea827ebc-7a9d-495a-ad7e-ffbbe3a96ee0, GlobSel=AssignType=Directly, SelType=Locally
    Button (870,100 150x30), "Setup Screen"
        OnMouseClick: FrameSelectionChange Selection=SelectedFrame=ea827ebc-7a9d-495a-ad7e-ffbbe3a96ee0, Selection=1, GlobSel=AssignType=Directly, SelType=Locally
    Button (870,150 150x30), "Alarms"
        OnMouseClick: FrameSelectionChange Selection=SelectedFrame=ea827ebc-7a9d-495a-ad7e-ffbbe3a96ee0, Selection=2, GlobSel=AssignType=Directly, SelType=Locally
    Button (870,200 150x30), "Manual Operations"
        OnMouseClick: FrameSelectionChange Selection=SelectedFrame=ea827ebc-7a9d-495a-ad7e-ffbbe3a96ee0, Selection=3, GlobSel=AssignType=Directly, SelType=Locally
    Ellipse (890,550 100x100), "RESET", invisible if: NOT :=MAIN.bStop
        OnMouseDown: toggle MAIN.bStop
    Ellipse (890,550 100x100), "STOP", invisible if: MAIN.bStop
        OnMouseDown: toggle MAIN.bStop
END_VISUALIZATION
